// TIA Portal project "Drivin_ a_3-phase_asynchronous_motor_from_different_points" (V15)

(* hardware
DEVICE "S7-1200 station_1"  S7-1200 Station
   slot 0: "Rack_0"  S7-1200 Rack  Rack  V1.0
   slot 1: "PLC_1"  CPU 1212C DC/DC/DC  6ES7 212-1AE40-0XB0  V4.2
*)

// ===== PLC "PLC_1"  CPU 1212C DC/DC/DC =====

VAR_GLOBAL   // PLC tag table "Default tag table"
   "I_THERMAL_RELAY" AT %I0.0 : Bool;
   "I_START_BTN_1" AT %I0.1 : Bool;
   "I_START_BTN_2" AT %I0.2 : Bool;
   "I_START_BTN_3" AT %I0.3 : Bool;
   "I_START_BTN_4" AT %I0.4 : Bool;
   "I_ESTOP" AT %I0.5 : Bool;
   "Q_MOTOR" AT %Q0.0 : Bool;
   "I_STOP_BTN_1" AT %I0.6 : Bool;
   "I_STOP_BTN_2" AT %I0.7 : Bool;
   "I_STOP_BTN_3" AT %I1.0 : Bool;
   "I_STOP_BTN_4" AT %I1.1 : Bool;
END_VAR

ORGANIZATION_BLOCK "Main"   // OB1, LAD, ProgramCycle
TITLE = "Main Program Sweep (Cycle)"
{ S7_Optimized_Access := 'TRUE' }
VERSION : 0.1
   VAR_INPUT
      Initial_Call : Bool;   // Initial call of this OB
      Remanence : Bool;   // =True, if remanent data are available
   END_VAR
BEGIN

REGION Network 1
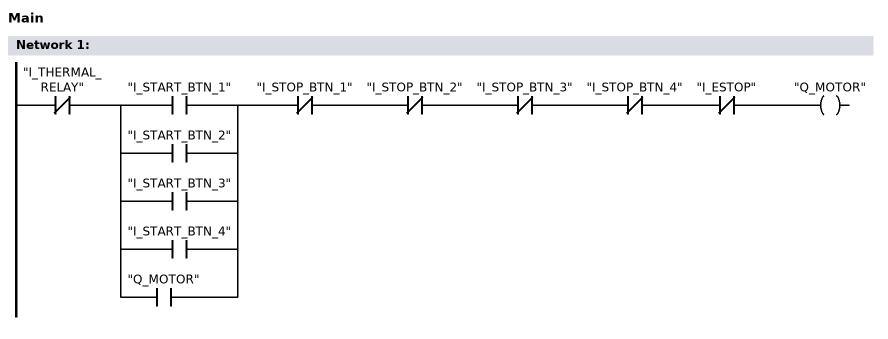
   RUNG wire#powerrail
      I_Contact( "I_THERMAL_RELAY" )
      wire#w1
      Contact( "I_START_BTN_1" )
      wire#w2
      I_Contact( "I_STOP_BTN_1" )
      I_Contact( "I_STOP_BTN_2" )
      I_Contact( "I_STOP_BTN_3" )
      I_Contact( "I_STOP_BTN_4" )
      I_Contact( "I_ESTOP" )
      Coil( "Q_MOTOR" )
   END_RUNG
   RUNG wire#w1
      Contact( "I_START_BTN_2" )
   END_RUNG wire#w2
   RUNG wire#w1
      Contact( "I_START_BTN_3" )
   END_RUNG wire#w2
   RUNG wire#w1
      Contact( "I_START_BTN_4" )
   END_RUNG wire#w2
   RUNG wire#w1
      Contact( "Q_MOTOR" )
   END_RUNG wire#w2
   // the same network as SCL:
   "Q_MOTOR" := NOT "I_THERMAL_RELAY" AND ("I_START_BTN_1" OR "I_START_BTN_2" OR "I_START_BTN_3" OR "I_START_BTN_4" OR "Q_MOTOR") AND NOT "I_STOP_BTN_1" AND NOT "I_STOP_BTN_2" AND NOT "I_STOP_BTN_3" AND NOT "I_STOP_BTN_4" AND NOT "I_ESTOP";
END_REGION
END_ORGANIZATION_BLOCK